//{attribute 'qualified_only'}
VAR_GLOBAL PERSISTENT
	OP80_DLY_BEF_MEAS : INT;
	OP80_VERT_SERVO_WORK_POS : REAL;
	OP80_VERT_SERVO_SFE_WORK_POS : REAL;	
END_VAR

(* stored: Version 1.1.0.1, ProductVersion 3.1.4024.11
   GVL OP80_Recipe: Id {736b295c-13c9-476b-ab47-e1a821ac25f3} *)
